// TwinCAT 3 PLC project Sample02
// ProgramVersion: 3.1.4022.4
// libraries:
//   Tc2_Standard, * (Beckhoff Automation GmbH)
//   Tc2_System, * (Beckhoff Automation GmbH)
//   Tc3_Module, * (Beckhoff Automation GmbH)
// project tree:
//   / ClassDiagram.TcCD (not stored), PlcTask.TcTTO
//   POUs/ FB_AmericanPizzaCalifornia.TcPOU, FB_AmericanPizzaMargherita.TcPOU, FB_AmericanPizzaNewYork.TcPOU, FB_ItalianPizzaMargherita.TcPOU, FB_ItalianPizzaMozzarella.TcPOU, FB_ItalianPizzaPiccante.TcPOU, FB_ItalianPizzaSalami.TcPOU, FB_PizzaAmericanStyle.TcPOU, FB_PizzaItalianStyle.TcPOU, I_Pizza.TcIO, MAIN.TcPOU
// real-time tasks:
//   TASK PlcTask: cycle T#10ms, priority 20, ADS port 350

CONFIGURATION Sample02
    RESOURCE PLC ON TwinCAT3
        TASK PlcTask(INTERVAL := T#10ms, PRIORITY := 20);
        PROGRAM MAIN WITH PlcTask : MAIN;
    END_RESOURCE
END_CONFIGURATION

// ---- POUs/I_Pizza.TcIO
INTERFACE I_Pizza

METHOD GetPrice : LREAL
VAR_INPUT
END_VAR
END_METHOD

END_INTERFACE

// ---- POUs/MAIN.TcPOU
PROGRAM MAIN
VAR
	fbItalianPizzaPiccante			: FB_ItalianPizzaPiccante;
	fbItalianPizzaMozzarella		: FB_ItalianPizzaMozzarella;
	fbItalianPizzaSalami			: FB_ItalianPizzaSalami;
	fbAmericanPizzaCalifornia		: FB_AmericanPizzaCalifornia;
	fbAmericanPizzaNewYork			: FB_AmericanPizzaNewYork;
	aPizza 							: ARRAY [1..5] OF I_Pizza;
	nIndex							: INT;
	lrPrice							: LREAL;
END_VAR

aPizza[1] := fbItalianPizzaPiccante;
aPizza[2] := fbItalianPizzaMozzarella;
aPizza[3] := fbItalianPizzaSalami;
aPizza[4] := fbAmericanPizzaCalifornia;
aPizza[5] := fbAmericanPizzaNewYork;

lrPrice := 0;
FOR nIndex := 1 TO 5 DO
	lrPrice := lrPrice + aPizza[nIndex].GetPrice();
END_FOR

END_PROGRAM

// ---- POUs/FB_ItalianPizzaPiccante.TcPOU
FUNCTION_BLOCK PUBLIC FB_ItalianPizzaPiccante EXTENDS FB_ItalianPizzaSalami
VAR_INPUT
END_VAR
VAR_OUTPUT
END_VAR
VAR
	bChilli		: BOOL := TRUE;
END_VAR

PROPERTY PUBLIC bHasChilli : BOOL
GET
bHasChilli := this^.bChilli;
END_GET
SET
this^.bChilli := bHasChilli;
END_SET
END_PROPERTY

METHOD PUBLIC GetPrice : LREAL
GetPrice := SUPER^.GetPrice();
IF (THIS^.bHasChilli) THEN
	GetPrice := GetPrice + 0.5;
END_IF
END_METHOD

END_FUNCTION_BLOCK

// ---- POUs/FB_ItalianPizzaSalami.TcPOU
FUNCTION_BLOCK PUBLIC FB_ItalianPizzaSalami EXTENDS FB_ItalianPizzaMargherita
VAR_INPUT
END_VAR
VAR_OUTPUT
END_VAR
VAR
	bSalami		: BOOL := TRUE;
END_VAR

PROPERTY PUBLIC bHasSalami : BOOL
GET
bHasSalami := this^.bSalami;
END_GET
SET
this^.bSalami := bHasSalami;
END_SET
END_PROPERTY

METHOD PUBLIC GetPrice : LREAL
GetPrice := SUPER^.GetPrice();
IF (THIS^.bSalami) THEN
	GetPrice := GetPrice + 1.4;
END_IF
END_METHOD

END_FUNCTION_BLOCK

// ---- POUs/FB_ItalianPizzaMargherita.TcPOU
FUNCTION_BLOCK PUBLIC FB_ItalianPizzaMargherita EXTENDS FB_PizzaItalianStyle
VAR_INPUT
END_VAR
VAR_OUTPUT
END_VAR
VAR
	bCheese		: BOOL := TRUE;
	bTomato		: BOOL := TRUE;
END_VAR

PROPERTY PUBLIC bHasCheese : BOOL
GET
bHasCheese := this^.bCheese;
END_GET
SET
this^.bCheese := bHasCheese;
END_SET
END_PROPERTY

PROPERTY PUBLIC bHasTomato : BOOL
GET
bHasTomato := this^.bTomato;
END_GET
SET
this^.bTomato := bHasTomato;
END_SET
END_PROPERTY

METHOD PUBLIC GetPrice : LREAL
GetPrice := SUPER^.GetPrice();
IF (THIS^.bCheese) THEN
	GetPrice := GetPrice + 1.1;
END_IF
IF (THIS^.bTomato) THEN
	GetPrice := GetPrice + 0.9;
END_IF
END_METHOD

END_FUNCTION_BLOCK

// ---- POUs/FB_PizzaItalianStyle.TcPOU
FUNCTION_BLOCK PUBLIC FB_PizzaItalianStyle IMPLEMENTS I_Pizza
VAR_INPUT
END_VAR
VAR_OUTPUT
END_VAR
VAR
END_VAR

METHOD PUBLIC GetPrice : LREAL
GetPrice := 4.5;
END_METHOD

END_FUNCTION_BLOCK

// ---- POUs/FB_ItalianPizzaMozzarella.TcPOU
FUNCTION_BLOCK PUBLIC FB_ItalianPizzaMozzarella EXTENDS FB_ItalianPizzaMargherita
VAR_INPUT
END_VAR
VAR_OUTPUT
END_VAR
VAR
	bBasil		: BOOL := TRUE;
END_VAR

PROPERTY PUBLIC bHasBasil : BOOL
GET
bHasBasil := this^.bBasil;
END_GET
SET
this^.bBasil := bHasBasil;
END_SET
END_PROPERTY

METHOD PUBLIC GetPrice : LREAL
GetPrice := SUPER^.GetPrice();
IF (THIS^.bBasil) THEN
	GetPrice := GetPrice + 0.25;
END_IF
END_METHOD

END_FUNCTION_BLOCK

// ---- POUs/FB_AmericanPizzaCalifornia.TcPOU
FUNCTION_BLOCK PUBLIC FB_AmericanPizzaCalifornia EXTENDS FB_AmericanPizzaMargherita
VAR_INPUT
END_VAR
VAR_OUTPUT
END_VAR
VAR
	bPepperoni	: BOOL := TRUE;
END_VAR

PROPERTY PUBLIC bHasPepperoni : BOOL
GET
bHasPepperoni := this^.bPepperoni;
END_GET
SET
this^.bPepperoni := bHasPepperoni;
END_SET
END_PROPERTY

METHOD PUBLIC GetPrice : LREAL
VAR_INPUT
END_VAR
GetPrice := SUPER^.GetPrice();
IF (THIS^.bPepperoni) THEN
	GetPrice := GetPrice + 0.4;
END_IF
END_METHOD

END_FUNCTION_BLOCK

// ---- POUs/FB_AmericanPizzaMargherita.TcPOU
FUNCTION_BLOCK PUBLIC FB_AmericanPizzaMargherita EXTENDS FB_PizzaAmericanStyle
VAR_INPUT
END_VAR
VAR_OUTPUT
END_VAR
VAR
	bCheese		: BOOL := TRUE;
	bTomato		: BOOL := TRUE;
END_VAR

PROPERTY PUBLIC bHasCheese : BOOL
GET
bHasCheese := this^.bCheese;
END_GET
SET
this^.bCheese := bHasCheese;
END_SET
END_PROPERTY

PROPERTY PUBLIC bHasTomato : BOOL
GET
bHasTomato := this^.bTomato;
END_GET
SET
this^.bTomato := bHasTomato;
END_SET
END_PROPERTY

METHOD PUBLIC GetPrice : LREAL
VAR_INPUT
END_VAR
GetPrice := SUPER^.GetPrice();
IF (THIS^.bCheese) THEN
	GetPrice := GetPrice + 1.1;
END_IF
IF (THIS^.bTomato) THEN
	GetPrice := GetPrice + 0.9;
END_IF
END_METHOD

END_FUNCTION_BLOCK

// ---- POUs/FB_PizzaAmericanStyle.TcPOU
FUNCTION_BLOCK PUBLIC FB_PizzaAmericanStyle IMPLEMENTS I_Pizza
VAR_INPUT
END_VAR
VAR_OUTPUT
END_VAR
VAR
END_VAR

METHOD PUBLIC GetPrice : LREAL
VAR_INPUT
END_VAR
GetPrice := 4.2;
END_METHOD

END_FUNCTION_BLOCK

// ---- POUs/FB_AmericanPizzaNewYork.TcPOU
FUNCTION_BLOCK PUBLIC FB_AmericanPizzaNewYork EXTENDS FB_AmericanPizzaMargherita
VAR_INPUT
END_VAR
VAR_OUTPUT
END_VAR
VAR
	bBroccoli	: BOOL := TRUE;
	bMushroom	: BOOL := TRUE;
END_VAR

PROPERTY PUBLIC bHasBroccoli : BOOL
GET
bHasBroccoli := this^.bBroccoli;
END_GET
SET
this^.bBroccoli := bHasBroccoli;
END_SET
END_PROPERTY

PROPERTY PUBLIC bHasMushroom : BOOL
GET
bHasMushroom := this^.bMushroom;
END_GET
SET
this^.bMushroom := bHasMushroom;
END_SET
END_PROPERTY

METHOD PUBLIC GetPrice : LREAL
VAR_INPUT
END_VAR
GetPrice := SUPER^.GetPrice();
IF (THIS^.bBroccoli) THEN
	GetPrice := GetPrice + 0.8;
END_IF
IF (THIS^.bMushroom) THEN
	GetPrice := GetPrice + 0.75;
END_IF
END_METHOD

END_FUNCTION_BLOCK
